# EPICS autosave request: iocBoot/iocValon5009/auto_settings_valon5009.req
file "valon5009_settings.req",                P=$(P),  R=$(R)
